TYPE ST_ITC_ZoneFlags :
(**************************************************************************************
 * 	Application		:	BoxControl Framework
 *	Revision		:	$Revision: 404529 $
 *	Revision date	:	$Date: 2018-04-23 08:21:38 +0200 (Mo., 23 Apr 2018) $
 *	Last changed by	:	$Author: b7bolm $
 *	URL				:	$URL: http://almscdc.swisslog.com/repo/SWPD/Development/BoxControlFramework/20_Release/trunk/01_Software/BCF/BCF/JumpStart/20_Product/10_App/12_E_Functions/10_Lib/10_Conv/01_DUTs/ST_ITC_ZoneFlags.TcDUT $
 *
 *	Purpose			:	Zone flags
 *
 * ------------------------------------------------------------------------------------
 *	Copyright Swisslog [IP AG], Switzerland. All rights reserved.
 * 
 * ------------------------------------------------------------------------------------
 *	
 * 	Revision History: 
 *
 * 	VERSION			DATE			INITIALS			DESCRIPTION
 *	0.1				01.01.2001		swl					Example
 *
 **************************************************************************************)	
STRUCT
	TransportTaksCompleteOccSent	: BOOL; // Store sent information
	TransportTaksCompleteSent		: BOOL; // Store sent information
	PositionClearSent				: BOOL; // Store sent information
	PositionOccupiedSent			: BOOL; // Store sent information
	IdentificationReportSent		: BOOL; // Store sent information
END_STRUCT
END_TYPE

(* stored: Version 1.1.0.1, ProductVersion 3.1.4022.12
   DUT ST_ITC_ZoneFlags: Id {87cf479e-5387-4caf-96ec-3504c3a8c3cb} *)
